FUNCTION_BLOCK ABSTRACT TaskBase EXTENDS ComponentBase IMPLEMENTS ITaskState
VAR
	i_taskBase : TaskBaseInternal;
END_VAR

METHOD Inihibits : BOOL
//This method is meant to be overriden
END_METHOD

METHOD newCommandState : BOOL
VAR_INPUT
	newTaskState : ENUM;
END_VAR
i_taskBase._newCommand := TRUE;
i_taskBase._state := newTaskState;
END_METHOD

{warning 'add property implementation'}
PROPERTY newTaskCommand : BOOL
GET
//newTaskCommand :=
END_GET
END_PROPERTY

METHOD Running : BOOL
VAR_INPUT
END_VAR
THIS^.Simulation();

IF newTaskCommand THEN

	IF taskReady THEN
		
		THIS^.Inihibits();
	
		THIS^.UpdateState();

	ELSE

		//REJECTED		

	END_IF
END_IF

THIS^.StateMachine();

THIS^.Cyclic();
END_METHOD

METHOD stateErrored : BOOL
VAR_INPUT
END_VAR
END_METHOD

METHOD stateFinished : BOOL
VAR_INPUT
END_VAR
i_taskBase._state := 0;
END_METHOD

METHOD StateMachine : BOOL
END_METHOD

//Ready indicates that the task is ready to accept commands
{attribute 'monitoring' := 'call'}
PROPERTY taskReady : BOOL
GET
taskReady := i_ComponentBase._ready;
END_GET
SET
i_ComponentBase._ready := taskReady;
END_SET
END_PROPERTY

//Gets the current state of the system
{attribute 'monitoring' := 'call'}
PROPERTY taskState : ENUM
GET

taskState := i_taskBase._state;
END_GET
END_PROPERTY

METHOD UpdateState : BOOL
END_METHOD

END_FUNCTION_BLOCK

(* stored: Version 1.1.0.1, ProductVersion 3.1.4024.12
   POU TaskBase: Id {11e525e0-645b-4df4-b2fb-22f19d8aff29}, SpecialFunc None
   Folder API: Id {fa7b63a7-59cf-4c12-b577-5e7473af5e23}
   Folder ApplicationOverrides: Id {38d144c6-40b6-4320-94ca-f6bb43b62195}
   Folder Internal: Id {0e960566-c110-4d07-93c2-d6c5d78d7f5f}
   Method Inihibits: Id {0087f8d2-5c7f-4a62-a915-5d55db385d44}
   Method newCommandState: Id {f0e11aaa-474a-41da-a433-67233cb55afc}
   Property newTaskCommand: Id {abd17dbf-36ab-4acf-9302-1631ffdd8ae9}
   Get Get: Id {25feb5aa-7b58-4fc7-a0d8-1a191cb27a01}
   Method Running: Id {fa085813-51d8-4282-8908-957f2a649b57}
   Method stateErrored: Id {a29a6bdc-8961-4e72-b5c8-9986d26c7307}
   Method stateFinished: Id {0e01e0bf-0d2f-48cf-a4a8-cac681f65a10}
   Method StateMachine: Id {8d58f681-a9ce-4bce-b521-193c540b10fe}
   Property taskReady: Id {700b7e26-f967-4e8d-8499-104188e09687}
   Get Get: Id {57e63903-3b80-4b15-831d-4bc339d57d54}
   Set Set: Id {b8cc81d5-fe59-44cc-bded-263742f9c532}
   Property taskState: Id {0037edbd-1327-4bd8-a4eb-83b875b0c5a7}
   Get Get: Id {f23eefa5-93ff-4b9e-be63-112cd0e9b4fa}
   Method UpdateState: Id {c750a4c5-92f0-4732-b52c-5a879b7774b7} *)
